FUNCTION_BLOCK Plant
  (* Standard: 61499-2 *)
  (* Version 0.1, 2015-00-10, syy, syy-PC *)
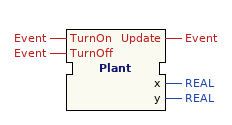
  EVENT_INPUT
    TurnOn;
    TurnOff;
  END_EVENT
  EVENT_OUTPUT
    Update;
  END_EVENT
  VAR_OUTPUT
    x : REAL;
    y : REAL;
  END_VAR
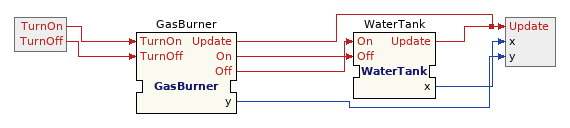
  FBS
    WaterTank : WaterTank;
    GasBurner : GasBurner;
  END_FBS
  EVENT_CONNECTIONS
    TurnOn TO GasBurner.TurnOn;
    TurnOff TO GasBurner.TurnOff;
    WaterTank.Update TO Update;
    GasBurner.Update TO Update;
    GasBurner.On TO WaterTank.On;
    GasBurner.Off TO WaterTank.Off;
  END_CONNECTIONS
  DATA_CONNECTIONS
    WaterTank.x TO x;
    GasBurner.y TO y;
  END_CONNECTIONS
END_FUNCTION_BLOCK
